FUNCTION_BLOCK FB_ProcessData
VAR_INPUT
	pd 				: 	REFERENCE TO ST_ProcessData;
END_VAR
VAR
	sensorRaw		:	ST_SensorRaw; 
END_VAR

(* Temperatur*)
pd.sensor.temperatureEvaporatingIn 		:=	RawToTemperature(sensorRaw.temperatureEvaporatingIn);
pd.sensor.temperatureEvaporatingOut 	:=	RawToTemperature(sensorRaw.temperatureEvaporatingOut);
pd.sensor.temperatureFlow 				:=	RawToTemperature(sensorRaw.temperatureFlow);
pd.sensor.temperatureReturn 			:=	RawToTemperature(sensorRaw.temperatureReturn);
pd.sensor.bufferTopTemperature 			:=	RawToTemperature(sensorRaw.bufferTopTemperature);
pd.sensor.bufferMiddleTemperature 		:=	RawToTemperature(sensorRaw.bufferMiddleTemperature);
pd.sensor.boilerTemperature				:=	RawToTemperature(sensorRaw.boilerTemperature);
pd.sensor.temperatureOverheatedGas 		:=	RawToTemperature(sensorRaw.temperatureOverheatedGas);
pd.sensor.temperatureEvaporatingIn 		:=	RawToTemperature(sensorRaw.temperatureEvaporatingIn);
pd.sensor.temperatureEvaporatingIn 		:=	RawToTemperature(sensorRaw.temperatureEvaporatingIn);
pd.sensor.temperatureEvaporatingIn 		:=	RawToTemperature(sensorRaw.temperatureEvaporatingIn);

(* Pressure Difference im mBar -  0-10 Volt  or  -10V to +10V *)
pd.sensor.pressureDifferenceEvaporator	:= 	RawToRealAnalog(sensorRaw.pressureDifferenceEvaporator, 0, 200, 10);

(* Pressure in Bar - using 4-20mmA Sensors*)
pd.sensor.pressureHigh	:= 	RawToRealAnalog(sensorRaw.pressureHigh, 0, 18, 10);			(* Range from 0 to 18.0 bar *)
pd.sensor.pressureLow	:= 	RawToRealAnalog(sensorRaw.pressureLow, -0.5, 7, 10);		(* Range from -0.5 to 7.0 bar *)

METHOD RawToRealAnalog : REAL
VAR_INPUT
	rawVal		: INT;
	rawMin		: REAL;
	rawMax		: REAL;	
	roundFactor	: INT;
END_VAR
VAR CONSTANT
	highValue 	: INT := 16#7FFF;  // Hexadezimale Zahl 0x7FFF
END_VAR
VAR
	realVal		: REAL;
END_VAR
realVal := ((rawMax - rawMin) * rawVal) / highValue + rawMin;
RawToRealAnalog := ScaleAndRound(realVal, roundFactor);
END_METHOD

METHOD INTERNAL RawToTemperature : REAL
VAR_INPUT
	raw : INT;
END_VAR
RawToTemperature :=  (INT_TO_REAL (raw)) / 10;
END_METHOD

END_FUNCTION_BLOCK

(* stored: Version 1.1.0.1
   POU FB_ProcessData: Id {8d629261-798f-4877-9443-8dbcc04e3ba2}, SpecialFunc None
   Method RawToRealAnalog: Id {355a4604-1918-414d-9adf-7ec3cdd623de}
   Method RawToTemperature: Id {8cedd837-1386-413c-9ce0-3d1e6ffcbdd0} *)
